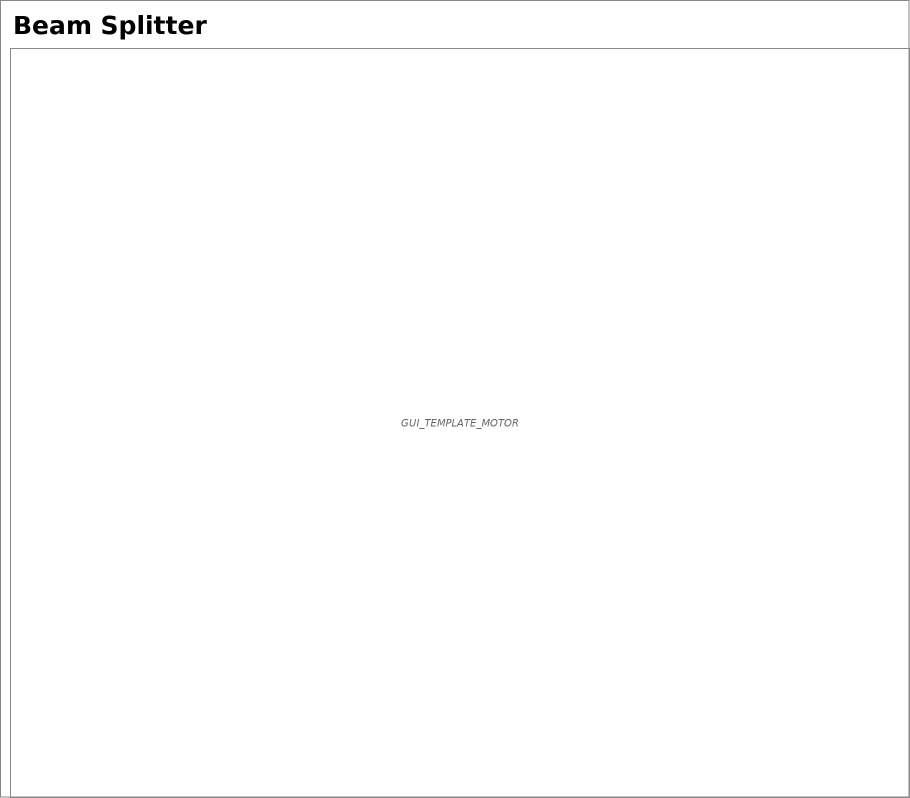
VISUALIZATION VISU_HMI_BEAM_SPLITTER  // 910x798
    Label (10,10 199x30), "Beam Splitter"
    Frame (10,48 900x750)
        shows GUI_TEMPLATE_MOTOR(m_Instance := MAIN.nott_ics.Calibration_Unit_Beam_Splitter.NBS)
END_VISUALIZATION

(* stored: Version 1.1.0.1, ProductVersion 3.1.4024.14
   Visu VISU_HMI_BEAM_SPLITTER: Id {ffaa4b80-4a22-4ce0-9c5b-6f9bcc8bed52} *)
